{attribute 'TcGenerated'}
{attribute 'no-analysis'}
{attribute 'linkalways'}
// This function has been automatically generated from the project information.
VAR_GLOBAL CONSTANT
	{attribute 'const_non_replaced'}
	stLibVersion_AdsGamepad : ST_LibVersion := (iMajor := 2, iMinor := 2, iBuild := 1, iRevision := 0, nFlags := 1, sVersion := '2.2.1');
END_VAR

(* stored: Version 1.1.0.1, ProductVersion 3.1.4026.18
   GVL Global_Version: Id {3c93b8be-b8b7-087a-25e9-302e5728b21a} *)
